// TwinCAT 3 PLC project PLC
// ProgramVersion: 3.1.4026.17
// libraries:
//   Tc2_Standard, * (Beckhoff Automation GmbH)
//   Tc2_System, * (Beckhoff Automation GmbH)
//   Tc2_Utilities, * (Beckhoff Automation GmbH)
// project tree:
//   Application Arguments/ AxisArgument.TcPOU, TemperatureArgument.TcPOU
//   GVLs/ GVL.TcGVL
//   Logging/Interfaces/ I_Base.TcIO, I_SimpleLocalLogger.TcIO, I_SimpleLogArgument.TcIO, I_SimpleLogger.TcIO, I_SimpleLogMessage.TcIO, I_SimpleLogPublisher.TcIO, I_SimpleLogSource.TcIO, I_ToString.TcIO
//   Logging/ SimpleLog.TcPOU, SimpleLocalLogger.TcPOU, SimpleLogMessage.TcPOU, SimpleLogSource.TcPOU
//   / MAIN.TcPOU, Parameters.TcGVL, PlcTask.TcTTO
// real-time tasks:
//   TASK PlcTask: cycle T#10ms, priority 20, ADS port 350

CONFIGURATION PLC
    RESOURCE PLC ON TwinCAT3
        TASK PlcTask(INTERVAL := T#10ms, PRIORITY := 20);
        PROGRAM MAIN WITH PlcTask : MAIN;
    END_RESOURCE
END_CONFIGURATION

// ---- GVLs/GVL.TcGVL
{attribute 'qualified_only'}
VAR_GLOBAL
	Logger		: SimpleLog<2>;
END_VAR

// ---- Parameters.TcGVL
{attribute 'qualified_only'}
VAR_GLOBAL CONSTANT
	MaxMessages : USINT := 10;
END_VAR

// ---- Logging/Interfaces/I_Base.TcIO
INTERFACE I_Base EXTENDS __SYSTEM.IQUERYINTERFACE

END_INTERFACE

// ---- Logging/Interfaces/I_SimpleLocalLogger.TcIO
INTERFACE I_SimpleLocalLogger EXTENDS I_Base, I_SimpleLogger

PROPERTY Messages : REFERENCE TO ARRAY[0..Parameters.MaxMessages - 1] OF T_MaxString
GET
END_GET
END_PROPERTY

END_INTERFACE

// ---- Logging/Interfaces/I_SimpleLogArgument.TcIO
INTERFACE I_SimpleLogArgument EXTENDS I_Base,I_ToString

END_INTERFACE

// ---- Logging/Interfaces/I_SimpleLogger.TcIO
INTERFACE I_SimpleLogger EXTENDS I_Base

METHOD LogMessage
VAR_INPUT
	Source	  : I_SimpleLogSource;
	Message	  : I_SimpleLogMessage;
	Argument : I_SimpleLogArgument := 0;
END_VAR
END_METHOD

END_INTERFACE

// ---- Logging/Interfaces/I_SimpleLogMessage.TcIO
INTERFACE I_SimpleLogMessage EXTENDS I_Base

{attribute 'monitoring':='call'}
PROPERTY Message : T_MaxString
GET
END_GET
END_PROPERTY

{attribute 'monitoring':='call'}
PROPERTY Severity : USINT
GET
END_GET
END_PROPERTY

END_INTERFACE

// ---- Logging/Interfaces/I_SimpleLogPublisher.TcIO
INTERFACE I_SimpleLogPublisher EXTENDS I_Base

METHOD Subscribe
VAR_INPUT
	Logger : I_SimpleLogger;
END_VAR
END_METHOD

END_INTERFACE

// ---- Logging/Interfaces/I_SimpleLogSource.TcIO
INTERFACE I_SimpleLogSource EXTENDS I_Base

{attribute 'monitoring':='call'}
PROPERTY SourceName : T_MaxString
GET
END_GET
END_PROPERTY

{attribute 'monitoring':='call'}
PROPERTY TimeStamp : T_FILETIME64
GET
END_GET
END_PROPERTY

END_INTERFACE

// ---- Logging/Interfaces/I_ToString.TcIO
INTERFACE I_ToString EXTENDS I_Base

METHOD ToString : T_MaxString
VAR_INPUT
END_VAR
END_METHOD

END_INTERFACE

// ---- MAIN.TcPOU
PROGRAM MAIN
VAR
	State				: USINT;
	LocalLogger			: SimpleLocalLogger;
	Message				: SimpleLogMessage;
	Source				: SimpleLogSource;
	LogAMessage			: BOOL;
	IndividualMessage	: BOOL;
	ArgumentExample		: BOOL;
	TemperatureArgument : TemperatureArgument;
	AxisArgument		: AxisArgument;
END_VAR

CASE State OF
	0:
		GVL.Logger.Subscribe(LocalLogger);
		State := 10;

	10:
END_CASE

IF LogAMessage THEN
	LogAMessage := FALSE;
	GVL.Logger.LogMessage(Source, Message);
END_IF

IF IndividualMessage THEN
	IndividualMessage := FALSE;
	GVL.Logger.LogMessageIndividual(Message := 'My Individual Message');
END_IF

IF ArgumentExample THEN
	ArgumentExample						  := FALSE;
	TemperatureArgument.ActualTemperature := 50.1;
	TemperatureArgument.SetPoint		  := 50.2;
	Message.Message						  := 'Actual within tolerance.';
	GVL.Logger.LogMessage(Source, Message, TemperatureArgument);
	AxisArgument.Position	  := 123.5;
	AxisArgument.Velocity	  := 300;
	AxisArgument.Acceleration := -100;
	AxisArgument.Deceleration := 100;
	Message.Message			  := 'Acceleration outside of limits.';
	GVL.Logger.LogMessage(Source, Message, AxisArgument);
END_IF

END_PROGRAM

// ---- Logging/SimpleLocalLogger.TcPOU
FUNCTION_BLOCK SimpleLocalLogger IMPLEMENTS I_SimpleLocalLogger
VAR
	{attribute 'hide'}
	_Messages	 : ARRAY[0..Parameters.MaxMessages - 1] OF T_MaxString;
	{attribute 'hide'}
	CurrentIndex : USINT;
END_VAR

METHOD LogMessage
VAR_INPUT
	Source	 : I_SimpleLogSource;
	Message	 : I_SimpleLogMessage;
	Argument : I_SimpleLogArgument := 0;
END_VAR

VAR
	TimeStamp  : T_FILETIME64;
	TimeString : T_MaxString;
END_VAR
IF Source.TimeStamp = 0 THEN
	TimeStamp  := F_GetSystemTime();
	TimeString := SYSTEMTIME_TO_STRING(FILETIME64_TO_SYSTEMTIME(TimeStamp));
END_IF

_Messages[CurrentIndex] := CONCAT(TimeString, CONCAT(' ', CONCAT(Source.SourceName, CONCAT(': ', Message.Message))));
IF Argument <> 0 THEN
	_Messages[CurrentIndex] := CONCAT(_Messages[CurrentIndex], CONCAT(' : ', Argument.ToString()));
END_IF

CurrentIndex := CurrentIndex + 1;
IF CurrentIndex = Parameters.MaxMessages THEN
	CurrentIndex := 0;
END_IF
END_METHOD

{attribute 'monitoring' := 'call'}
PROPERTY Messages : REFERENCE TO ARRAY[0..Parameters.MaxMessages - 1] OF T_MaxString
GET
Messages REF= _Messages;
END_GET
END_PROPERTY

END_FUNCTION_BLOCK

// ---- Logging/SimpleLogMessage.TcPOU
FUNCTION_BLOCK SimpleLogMessage IMPLEMENTS I_SimpleLogMessage
VAR
	{attribute 'hide'}
	_Message : T_MaxString;
	{attribute 'hide'}
	_Severity : USINT;
END_VAR

{attribute 'monitoring' := 'call'}
PROPERTY Message : T_MaxString
GET
Message := _Message;
END_GET
SET
_Message := Message;
END_SET
END_PROPERTY

{attribute 'monitoring' := 'call'}
PROPERTY Severity : USINT
GET
Severity := _Severity;
END_GET
SET
_Severity := Severity;
END_SET
END_PROPERTY

END_FUNCTION_BLOCK

// ---- Logging/SimpleLogSource.TcPOU
FUNCTION_BLOCK SimpleLogSource IMPLEMENTS I_SimpleLogSource
VAR
	{attribute 'hide'}
	_SourceName : T_MaxString;
	{attribute 'hide'}
	_TimeStamp : T_FILETIME64;
END_VAR

{attribute 'monitoring' := 'call'}
PROPERTY SourceName : T_MaxString
GET
SourceName := _SourceName;
END_GET
SET
_SourceName := SourceName;
END_SET
END_PROPERTY

{attribute 'monitoring' := 'call'}
PROPERTY TimeStamp : T_FILETIME64
GET
TimeStamp := _TimeStamp;
END_GET
SET
_TimeStamp := TimeStamp;
END_SET
END_PROPERTY

END_FUNCTION_BLOCK

// ---- Application Arguments/TemperatureArgument.TcPOU
{attribute 'hide_all_locals'}
FUNCTION_BLOCK TemperatureArgument IMPLEMENTS I_SimpleLogArgument
VAR
	_SetPoint : LREAL;
	_Actual	  : LREAL;
END_VAR

{attribute 'monitoring':='call'}
PROPERTY ActualTemperature : LREAL
GET
ActualTemperature := _Actual;
END_GET
SET
_Actual := ActualTemperature;
END_SET
END_PROPERTY

{attribute 'monitoring':='call'}
PROPERTY SetPoint : LREAL
GET
SetPoint := _SetPoint;
END_GET
SET
_SetPoint := SetPoint;
END_SET
END_PROPERTY

METHOD ToString : T_MaxString
ToString := Concat('Set Temperature: ', CONCAT(TO_STRING(_SetPoint), CONCAT(' , Actual Temp: ', TO_STRING(_Actual))));
END_METHOD

END_FUNCTION_BLOCK

// ---- Application Arguments/AxisArgument.TcPOU
{attribute 'hide_all_locals'}
FUNCTION_BLOCK AxisArgument IMPLEMENTS I_SimpleLogArgument
VAR
	_Position	  : LREAL;
	_Velocity	  : LREAL;
	_Acceleration : LREAL;
	_Deceleration : LREAL;
END_VAR

{attribute 'monitoring':='call'}
PROPERTY Acceleration : LREAL
GET
Acceleration := _Acceleration;
END_GET
SET
_Acceleration := Acceleration;
END_SET
END_PROPERTY

{attribute 'monitoring':='call'}
PROPERTY Deceleration : LREAL
GET
Deceleration := _Deceleration;
END_GET
SET
_Deceleration := Deceleration;
END_SET
END_PROPERTY

{attribute 'monitoring':='call'}
PROPERTY Position : LREAL
GET
Position := _Position;
END_GET
SET
_Position := Position;
END_SET
END_PROPERTY

METHOD ToString : T_MaxString
ToString :=
	Concat('Pos: ',
		   CONCAT(TO_STRING(_Position), CONCAT(' , Vel: ', CONCAT(TO_STRING(_Velocity), CONCAT(' , Accel: ', CONCAT(TO_STRING(_Acceleration), CONCAT(' , Decel: ', TO_STRING(_Deceleration))))))));
END_METHOD

{attribute 'monitoring':='call'}
PROPERTY Velocity : LREAL
GET
Velocity := _Velocity;
END_GET
SET
_Velocity := Velocity;
END_SET
END_PROPERTY

END_FUNCTION_BLOCK

// ---- Logging/SimpleLog.TcPOU
FUNCTION_BLOCK SimpleLog
VAR_GENERIC CONSTANT
	NumberOfSubscribers : USINT := 5;
END_VAR
 
IMPLEMENTS I_SimpleLogPublisher, I_SimpleLogger
VAR
	SubscriberCount : USINT;
	_Subscribers : ARRAY[0..NumberOfSubscribers - 1] OF I_SimpleLogger;
END_VAR

METHOD LogMessage
VAR_INPUT
	Source	 : I_SimpleLogSource;
	Message	 : I_SimpleLogMessage;
	Argument : I_SimpleLogArgument := 0;
END_VAR

VAR
	i : UDINT;
END_VAR
FOR i := 0 TO NumberOfSubscribers - 1 DO
	IF _Subscribers[i] = 0 THEN
		CONTINUE;
	END_IF

	_Subscribers[i].LogMessage(Source, Message, Argument);
END_FOR
END_METHOD

METHOD LogMessageIndividual
VAR_INPUT
	TimeStamp  : T_FILETIME64 := 0;
	SourceName : T_MaxString  := '';
	Severity   : USINT		  := 0;
	Message	   : T_MaxString;
END_VAR

VAR
	LogSource	: SimpleLogSource;
	LogMessage : SimpleLogMessage;
END_VAR
LogSource.TimeStamp	 := TimeStamp;
LogSource.SourceName := SourceName;
LogMessage.Severity	 := Severity;
LogMessage.Message	 := Message;
THIS^.LogMessage(LogSource, LogMessage);
END_METHOD

METHOD Subscribe
VAR_INPUT
	Logger : I_SimpleLogger;
END_VAR
IF SubscriberCount >= NumberOfSubscribers THEN
	RETURN;
END_IF

_Subscribers[SubscriberCount] := Logger;
SubscriberCount				  := SubscriberCount + 1;
END_METHOD

END_FUNCTION_BLOCK
